// TIA Portal V16 export
// export: Created 2025-12-18T09:29:15.1380624Z, ExportSetting WithDefaults, DisplayName Totally Integrated Automation Portal, DisplayVersion V16, DisplayName TIA Portal Version Control Interface, DisplayVersion V16, DisplayName TIA Portal Openness, DisplayVersion V16, DisplayName STEP 7 Professional, DisplayVersion V16, DisplayName STEP 7 Safety, DisplayVersion V16, DisplayName WinCC Advanced, DisplayVersion V16
FUNCTION_BLOCK "StationProcessControl"   // FB4, LAD
{ S7_Optimized_Access := 'TRUE' }
VERSION : 0.1
// stored: AutoNumber true, IsIECCheckEnabled false, IsRetainMemResEnabled false, MemoryReserve 100, SetENOAutomatically false, UDAEnableTagReadback false
   VAR_INPUT
      xPositionerSensor { ExternalAccessible := 'False'; ExternalVisible := 'False'; ExternalWritable := 'False'} : Bool;
      xClampSensor { ExternalAccessible := 'False'; ExternalVisible := 'False'; ExternalWritable := 'False'} : Bool;
      tProcessTime { ExternalAccessible := 'False'; ExternalVisible := 'False'; ExternalWritable := 'False'} : Time;
   END_VAR
   VAR_IN_OUT
      xPositionerClamp : Bool;
      xPositionerRaise : Bool;
      xInProcess : Bool;
      diProcessTimeLeft : DInt;
      xRequestData : Bool;
   END_VAR
   VAR
      xProcessDone : Bool := false;
      xEdgeMemory1 : Bool;
      xEdgeMemory2 : Bool := false;
      IEC_Timer_0_Instance { S7_SetPoint := 'True'} : TON_TIME;
   END_VAR
   VAR_TEMP   // added for the SCL form of the ladder/FBD networks
      _w1 : Bool;
   END_VAR
BEGIN

REGION Network 1: Clamp positioner if material is detected, request for data
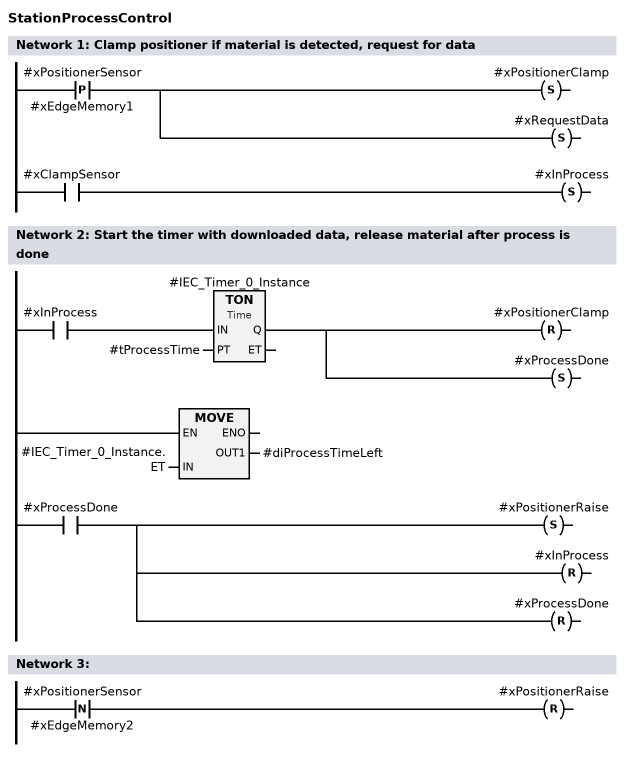
   RUNG wire#powerrail
      P_Contact(operand := #xPositionerSensor, bit := #xEdgeMemory1)
      wire#w1
      S_Coil( #xPositionerClamp )
   END_RUNG
   RUNG wire#w1
      S_Coil( #xRequestData )
   END_RUNG
   RUNG wire#powerrail
      Contact( #xClampSensor )
      S_Coil( #xInProcess )
   END_RUNG
   // the same network as SCL:
   #_w1 := #xPositionerSensor AND NOT #xEdgeMemory1;   // rising edge of #xPositionerSensor
   #xEdgeMemory1 := #xPositionerSensor;
   IF #_w1 THEN
       #xPositionerClamp := TRUE;
       #xRequestData := TRUE;
   END_IF;
   IF #xClampSensor THEN #xInProcess := TRUE; END_IF;
END_REGION

REGION Network 2: Start the timer with downloaded data, release material after process is done
   RUNG wire#powerrail
      Contact( #xInProcess )
      { S7_Templates := "time_type := Time" } #IEC_Timer_0_Instance.TON(pt := #tProcessTime, et =>)
      wire#w1
      R_Coil( #xPositionerClamp )
   END_RUNG
   RUNG wire#w1
      S_Coil( #xProcessDone )
   END_RUNG
   RUNG wire#powerrail
      Move(in := #IEC_Timer_0_Instance.ET, out1 => #diProcessTimeLeft)
   END_RUNG
   RUNG wire#powerrail
      Contact( #xProcessDone )
      wire#w2
      S_Coil( #xPositionerRaise )
   END_RUNG
   RUNG wire#w2
      R_Coil( #xInProcess )
   END_RUNG
   RUNG wire#w2
      R_Coil( #xProcessDone )
   END_RUNG
   // the same network as SCL:
   #IEC_Timer_0_Instance(IN := #xInProcess, PT := #tProcessTime);   // TON
   IF #IEC_Timer_0_Instance.Q THEN
       #xPositionerClamp := FALSE;
       #xProcessDone := TRUE;
   END_IF;
   #diProcessTimeLeft := #IEC_Timer_0_Instance.ET;
   IF #xProcessDone THEN
       #xPositionerRaise := TRUE;
       #xInProcess := FALSE;
       #xProcessDone := FALSE;
   END_IF;
END_REGION

REGION Network 3
   RUNG wire#powerrail
      N_Contact(operand := #xPositionerSensor, bit := #xEdgeMemory2)
      R_Coil( #xPositionerRaise )
   END_RUNG
   // the same network as SCL:
   #_w1 := NOT #xPositionerSensor AND #xEdgeMemory2;   // falling edge of #xPositionerSensor
   #xEdgeMemory2 := #xPositionerSensor;
   IF #_w1 THEN #xPositionerRaise := FALSE; END_IF;
END_REGION
END_FUNCTION_BLOCK
